{attribute 'qualified_only'}
VAR_GLOBAL
	// xDI%139.2_S1_2
	diNotAus_Kanal_A AT %I*: BOOL;
	// xDI%139.3_S1_2
	diNotAus_Kanal_B AT %I*: BOOL;
END_VAR

(* stored: Version 1.1.0.1, ProductVersion 3.1.4024.15
   GVL GVL: Id {528af200-5818-4f75-add0-cc3311a25bcf} *)
